(* CoDeSys 2.3 export: FB_CODE_FF70.EXP *)

(* POU PGN FB/FB_CODE_FF70, ST *)
FUNCTION_BLOCK FB_CODE_FF70 (*Torque / Speed Control*)
VAR_INPUT
	Enable   : BOOL;
	Source   : BYTE := 16#10;
	Priority : BYTE := 16#02;

	TaskTime     : WORD; (*PLC Taks Time (ms) eg: 10ms*)
	TransmitTime : WORD; (*Synchronous Transmision Time (ms) eg: 50ms*)

	PedalPerc  : REAL;
	PedalID    : BYTE;
	PedalFault : BOOL;
END_VAR
VAR_OUTPUT
	OUT : VARTYPE_EXTCANQUEUE;
	OUT_Enable : BOOL;
END_VAR
VAR
	TimeCnt : WORD;
	dwSrc   : DWORD;
	dwPty   : DWORD;

	bySpeedCtrl  : BYTE;
	byTorqueCtrl : BYTE;
END_VAR
IF Enable THEN
	TimeCnt := TimeCnt + TaskTime;

	IF TransmitTime <= TimeCnt THEN
		TimeCnt := 0;
		dwSrc   := Source;
		dwPty   := Priority AND 16#07;
		dwPty   := SHL( dwPty, 26 );

		REAL_TO_BUFFER( pBuffer:= ADR(OUT.rxData[0]), ByteSize := 2, Value:= PedalPerc, Scale:= 0.1, Offset := 0.0 );

		OUT.rxData[2] := PedalID;
		OUT.rxData[3] := 16#00;
		OUT.rxData[3].0 := PedalFault;
		OUT.rxData[4] := 16#00;
		OUT.rxData[5] := 16#00;
		OUT.rxData[6] := 16#00;
		OUT.rxData[7] := 16#00;

		OUT.length := 8;
		Out.cobId  := 16#80FF7000 OR dwSrc OR dwPty;
		OUT_Enable := TRUE;
	ELSE
		OUT_Enable := FALSE;

	END_IF
ELSE
	Out_Enable := FALSE;

END_IF
END_FUNCTION_BLOCK
